// TIA Portal V18 export
FUNCTION "AnaIn_Scaling" : Void   // FC5, FBD
TITLE = Analog Scaling of an Input
{ S7_Optimized_Access := 'TRUE' }
VERSION : 0.1
// -Normalize
// -Scale
// -OOR
// stored: AutoNumber true, IsIECCheckEnabled false, SetENOAutomatically false, UDAEnableTagReadback false
   VAR_INPUT
      IN_Int : DInt;   // Sensor Input Val usually PIWxxx
      IN_InputLowLim : Int;   // Min in from PIW sensor usually 0
      IN_InputHiLim : Int;   // Max in from PIW sensor usually 27648
      IN_ScaleMin : Real;   // Min value for the output scaling
      IN_ScaleMax : Real;   // Max value for the output scaling
   END_VAR
   VAR_OUTPUT
      Out_Real : Real;   // Scaled value
      Out_OOR : Bool;   // Out of Range
   END_VAR
   VAR_TEMP
      Out_norm : Real;
      Out_Scaled : Real;
      Dummy1 : Bool;
      Dummy2 : Bool;
   END_VAR
BEGIN

REGION Network 2 (SCL)
   IF #Dummy1 THEN
       #Dummy2 := FALSE;// Statement section IF

   END_IF;
END_REGION

REGION Network 3: HPU Proportional Valve: Normalize & Scaling of Input Feedback [+/-10V]
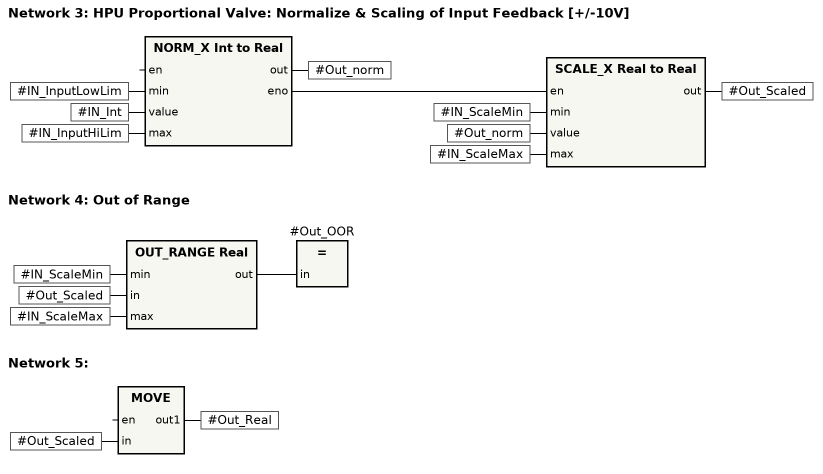
   #Out_norm := NORM_X(MIN := #IN_InputLowLim, VALUE := #IN_Int, MAX := #IN_InputHiLim);
   #Out_Scaled := SCALE_X(MIN := #IN_ScaleMin, VALUE := #Out_norm, MAX := #IN_ScaleMax);
END_REGION

REGION Network 4: Out of Range
   #Out_OOR := (#Out_Scaled < #IN_ScaleMin) OR (#Out_Scaled > #IN_ScaleMax);
END_REGION

REGION Network 5
   #Out_Real := #Out_Scaled;
END_REGION
END_FUNCTION
